INTERFACE ITF_Visitor

METHOD VisitBaseObject : BOOL
VAR_INPUT
	BaseObject : ITF_Base;
END_VAR
END_METHOD

END_INTERFACE

(* stored: Version 1.1.0.1, ProductVersion 3.1.4024.12
   Itf ITF_Visitor: Id {43d60605-6928-40db-819b-30d1104a5660}
   Method VisitBaseObject: Id {0a8d9862-8a42-4c31-9846-07c9a21e6996} *)
